{attribute addProperty BoxType "EL6851-0010-0016"}
{attribute addProperty Id "DMX_StatusAT %I*DMX_Status_CB89DD216480DMX_Channel_1_64AT %I*DMX_Channel_D03720FB512640WcStateAT %I*WcState_98A4DF7520.250InfoDataAT %I*InfoData_BC63D37F80100"}
{attribute addProperty CRC "2628321664"}
{attribute addProperty SizeInBites "658"}
{attribute addProperty SizeInBytes "82.25"}
TYPE EL6851_41B974CF :
STRUCT
	{attribute addProperty Name "DMX_Status"}
	DMX_Status : DMX_Status_CB89DD21;
	{attribute addProperty Name "DMX_Channel_1_64"}
	DMX_Channel_1_64 : DMX_Channel_D03720FB;
	{attribute addProperty Name "WcState"}
	WcState : WcState_98A4DF75;
	{attribute addProperty Name "InfoData"}
	InfoData : InfoData_BC63D37F;
END_STRUCT
END_TYPE

(* stored: Version 1.2.0.0, ProductVersion 3.1.4024.9
   DUT EL6851_41B974CF: Id {0fb10b08-92dc-4cc7-a9d2-eed4c8f8e23c} *)
